INTERFACE I_Fallible


METHOD GetError : BOOL
END_METHOD


METHOD GetErrorMsg : T_MaxString
END_METHOD

END_INTERFACE

(* stored: Version 1.1.0.1
   Itf I_Fallible: Id {1f0d17b4-8afe-43af-a630-1d3684ca167f}
   Method GetError: Id {12a6abc9-7d4a-4820-bf65-1b5eb91442ba}
   Method GetErrorMsg: Id {5723660d-5329-4105-9756-0ce30eca9d55} *)
